// TIA Portal V17 export
// export: Created 2025-03-10T13:12:15.9920924Z, ExportSetting WithDefaults, DisplayName Totally Integrated Automation Portal, DisplayVersion V17 Update 8, DisplayName TIA Portal Openness, DisplayVersion V17 Update 8, DisplayName TIA Portal Version Control Interface, DisplayVersion V17, DisplayName SINAMICS Startdrive Advanced, DisplayVersion V17 SP2, DisplayName SINAMICS Startdrive G110M, G120, G120C, G120D, G120P, G115D, DisplayVersion V17 SP2, DisplayName SINAMICS Startdrive G130, G150, S120, S150, SINAMICS MV, S210, DisplayVersion V17 SP2, DisplayName STEP 7 Professional, DisplayVersion V17 Update 8, DisplayName SINUMERIK ONE STEP 7 Toolbox, DisplayVersion V17 Update 12, DisplayName SINUMERIK 840D sl STEP 7 Toolbox, DisplayVersion V17 Update 12, DisplayName STEP 7 Safety, DisplayVersion V17 Update 6, DisplayName WinCC Advanced, DisplayVersion V17 Update 8
TYPE "READ_WRITE_DATA"
// stored: IsFailsafeCompliant false
   STRUCT
      IO_field : Array[0..79] of Bool;
      SoftkeyLeft0 : Bool;
      SoftkeyLeft1 : Bool;
      SoftkeyLeft2 : Bool;
      SoftkeyLeft3 : Bool;
      SoftkeyLeft4 : Bool;
      SoftkeyLeft5 : Bool;
      SoftkeyLeft6 : Bool;
      Page_up : Bool;
      SoftkeyRight0 : Bool;
      SoftkeyRight1 : Bool;
      SoftkeyRight2 : Bool;
      SoftkeyRight3 : Bool;
      SoftkeyRight4 : Bool;
      SoftkeyRight5 : Bool;
      SoftkeyRight6 : Bool;
      Page_Down : Bool;
      Pushbutton : Array[12..21] of Byte;
   END_STRUCT;
END_TYPE
